# EPICS autosave request: iocBoot/ioc13idd_micromax2/auto_settings.req
file "roper_settings.req",        P=$(P),  R=cam1:
file "NDStdArrays_settings.req",  P=$(P),  R=image1:
file "commonPlugin_settings.req",  P=$(P)
